(* CODESYS project IndraLogic.project

Project tree, tasks and I/O mapping:
  IndraMotionMlc1 : IndraControl XM2, Bosch Rexroth AG, order no. dependent on customer specific configuration, version 14.22.36.0
    application Application
      libraries: Linked List, 1.2.1.14 (Bosch Rexroth); MQTT Client, 2.3.8.14 (Bosch Rexroth)
      task PlcTask (cyclic, interval 10 ms, priority 5, watchdog 10 ms x 2) calls PlcProg
      task MotionTask (externalevent, external event EVENT_OP_MODE_MOTION_CYCLIC, priority 2, watchdog 4000 µs x 1) calls MotionProg
      function CheckBounds [ST]
      Symbols
      program PlcProg [ST]
      program MotionProg [ST]
      global variables MlcVarGlobal
      global variables IO
    S20_I_O : S20_I_O, Bosch Rexroth AG, version 14.22.10.1
    Sercos_III_Master : SercosIII Master, Rexroth, order no. 1, version 14.6.0.0
*)

// IndraMotionMlc1/Application/MlcVarGlobal
(* Automatically generated code by XLC/MLC. *)
(* Please don't edit, the code will be overwritten. For usercode use UserVarGlobal! *)
{attribute 'linkalways'}
{attribute 'analysis' := '-33'}
VAR_GLOBAL CONSTANT

(*Real axis "Axis1" with axis number 2*)
Axis1: AXIS_REF :=(CntrlNo:=LOCAL_CNTRL,AxisNo:=AXIS_2);


(*Probe 001*)
TouchProbe001: TOUCHPROBE_REF :=(CntrlNo:=LOCAL_CNTRL,TouchProbeNo:=TOUCHPROBE_1);

(*Probe 002*)
TouchProbe002: TOUCHPROBE_REF :=(CntrlNo:=LOCAL_CNTRL,TouchProbeNo:=TOUCHPROBE_2);

(*Probe 003*)
TouchProbe003: TOUCHPROBE_REF :=(CntrlNo:=LOCAL_CNTRL,TouchProbeNo:=TOUCHPROBE_3);

(*Probe 004*)
TouchProbe004: TOUCHPROBE_REF :=(CntrlNo:=LOCAL_CNTRL,TouchProbeNo:=TOUCHPROBE_4);

(*Probe 005*)
TouchProbe005: TOUCHPROBE_REF :=(CntrlNo:=LOCAL_CNTRL,TouchProbeNo:=TOUCHPROBE_5);

(*Probe 006*)
TouchProbe006: TOUCHPROBE_REF :=(CntrlNo:=LOCAL_CNTRL,TouchProbeNo:=TOUCHPROBE_6);

(*Probe 007*)
TouchProbe007: TOUCHPROBE_REF :=(CntrlNo:=LOCAL_CNTRL,TouchProbeNo:=TOUCHPROBE_7);

(*Probe 008*)
TouchProbe008: TOUCHPROBE_REF :=(CntrlNo:=LOCAL_CNTRL,TouchProbeNo:=TOUCHPROBE_8);

(*Probe 009*)
TouchProbe009: TOUCHPROBE_REF :=(CntrlNo:=LOCAL_CNTRL,TouchProbeNo:=TOUCHPROBE_9);

(*Probe 010*)
TouchProbe010: TOUCHPROBE_REF :=(CntrlNo:=LOCAL_CNTRL,TouchProbeNo:=TOUCHPROBE_10);

(*Probe 011*)
TouchProbe011: TOUCHPROBE_REF :=(CntrlNo:=LOCAL_CNTRL,TouchProbeNo:=TOUCHPROBE_11);

(*Probe 012*)
TouchProbe012: TOUCHPROBE_REF :=(CntrlNo:=LOCAL_CNTRL,TouchProbeNo:=TOUCHPROBE_12);

(*Probe 013*)
TouchProbe013: TOUCHPROBE_REF :=(CntrlNo:=LOCAL_CNTRL,TouchProbeNo:=TOUCHPROBE_13);

(*Probe 014*)
TouchProbe014: TOUCHPROBE_REF :=(CntrlNo:=LOCAL_CNTRL,TouchProbeNo:=TOUCHPROBE_14);

(*Probe 015*)
TouchProbe015: TOUCHPROBE_REF :=(CntrlNo:=LOCAL_CNTRL,TouchProbeNo:=TOUCHPROBE_15);

(*Probe 016*)
TouchProbe016: TOUCHPROBE_REF :=(CntrlNo:=LOCAL_CNTRL,TouchProbeNo:=TOUCHPROBE_16);

(*Probe 017*)
TouchProbe017: TOUCHPROBE_REF :=(CntrlNo:=LOCAL_CNTRL,TouchProbeNo:=TOUCHPROBE_17);

(*Probe 018*)
TouchProbe018: TOUCHPROBE_REF :=(CntrlNo:=LOCAL_CNTRL,TouchProbeNo:=TOUCHPROBE_18);

(*Probe 019*)
TouchProbe019: TOUCHPROBE_REF :=(CntrlNo:=LOCAL_CNTRL,TouchProbeNo:=TOUCHPROBE_19);

(*Probe 020*)
TouchProbe020: TOUCHPROBE_REF :=(CntrlNo:=LOCAL_CNTRL,TouchProbeNo:=TOUCHPROBE_20);

(*Probe 021*)
TouchProbe021: TOUCHPROBE_REF :=(CntrlNo:=LOCAL_CNTRL,TouchProbeNo:=TOUCHPROBE_21);

(*Probe 022*)
TouchProbe022: TOUCHPROBE_REF :=(CntrlNo:=LOCAL_CNTRL,TouchProbeNo:=TOUCHPROBE_22);

(*Probe 023*)
TouchProbe023: TOUCHPROBE_REF :=(CntrlNo:=LOCAL_CNTRL,TouchProbeNo:=TOUCHPROBE_23);

(*Probe 024*)
TouchProbe024: TOUCHPROBE_REF :=(CntrlNo:=LOCAL_CNTRL,TouchProbeNo:=TOUCHPROBE_24);

(*Probe 025*)
TouchProbe025: TOUCHPROBE_REF :=(CntrlNo:=LOCAL_CNTRL,TouchProbeNo:=TOUCHPROBE_25);

(*Probe 026*)
TouchProbe026: TOUCHPROBE_REF :=(CntrlNo:=LOCAL_CNTRL,TouchProbeNo:=TOUCHPROBE_26);

(*Probe 027*)
TouchProbe027: TOUCHPROBE_REF :=(CntrlNo:=LOCAL_CNTRL,TouchProbeNo:=TOUCHPROBE_27);

(*Probe 028*)
TouchProbe028: TOUCHPROBE_REF :=(CntrlNo:=LOCAL_CNTRL,TouchProbeNo:=TOUCHPROBE_28);

(*Probe 029*)
TouchProbe029: TOUCHPROBE_REF :=(CntrlNo:=LOCAL_CNTRL,TouchProbeNo:=TOUCHPROBE_29);

(*Probe 030*)
TouchProbe030: TOUCHPROBE_REF :=(CntrlNo:=LOCAL_CNTRL,TouchProbeNo:=TOUCHPROBE_30);

(*Probe 031*)
TouchProbe031: TOUCHPROBE_REF :=(CntrlNo:=LOCAL_CNTRL,TouchProbeNo:=TOUCHPROBE_31);

(*Probe 032*)
TouchProbe032: TOUCHPROBE_REF :=(CntrlNo:=LOCAL_CNTRL,TouchProbeNo:=TOUCHPROBE_32);

(*Probe 033*)
TouchProbe033: TOUCHPROBE_REF :=(CntrlNo:=LOCAL_CNTRL,TouchProbeNo:=TOUCHPROBE_33);

(*Probe 034*)
TouchProbe034: TOUCHPROBE_REF :=(CntrlNo:=LOCAL_CNTRL,TouchProbeNo:=TOUCHPROBE_34);

(*Probe 035*)
TouchProbe035: TOUCHPROBE_REF :=(CntrlNo:=LOCAL_CNTRL,TouchProbeNo:=TOUCHPROBE_35);

(*Probe 036*)
TouchProbe036: TOUCHPROBE_REF :=(CntrlNo:=LOCAL_CNTRL,TouchProbeNo:=TOUCHPROBE_36);

(*Probe 037*)
TouchProbe037: TOUCHPROBE_REF :=(CntrlNo:=LOCAL_CNTRL,TouchProbeNo:=TOUCHPROBE_37);

(*Probe 038*)
TouchProbe038: TOUCHPROBE_REF :=(CntrlNo:=LOCAL_CNTRL,TouchProbeNo:=TOUCHPROBE_38);

(*Probe 039*)
TouchProbe039: TOUCHPROBE_REF :=(CntrlNo:=LOCAL_CNTRL,TouchProbeNo:=TOUCHPROBE_39);

(*Probe 040*)
TouchProbe040: TOUCHPROBE_REF :=(CntrlNo:=LOCAL_CNTRL,TouchProbeNo:=TOUCHPROBE_40);

(*Probe 041*)
TouchProbe041: TOUCHPROBE_REF :=(CntrlNo:=LOCAL_CNTRL,TouchProbeNo:=TOUCHPROBE_41);

(*Probe 042*)
TouchProbe042: TOUCHPROBE_REF :=(CntrlNo:=LOCAL_CNTRL,TouchProbeNo:=TOUCHPROBE_42);

(*Probe 043*)
TouchProbe043: TOUCHPROBE_REF :=(CntrlNo:=LOCAL_CNTRL,TouchProbeNo:=TOUCHPROBE_43);

(*Probe 044*)
TouchProbe044: TOUCHPROBE_REF :=(CntrlNo:=LOCAL_CNTRL,TouchProbeNo:=TOUCHPROBE_44);

(*Probe 045*)
TouchProbe045: TOUCHPROBE_REF :=(CntrlNo:=LOCAL_CNTRL,TouchProbeNo:=TOUCHPROBE_45);

(*Probe 046*)
TouchProbe046: TOUCHPROBE_REF :=(CntrlNo:=LOCAL_CNTRL,TouchProbeNo:=TOUCHPROBE_46);

(*Probe 047*)
TouchProbe047: TOUCHPROBE_REF :=(CntrlNo:=LOCAL_CNTRL,TouchProbeNo:=TOUCHPROBE_47);

(*Probe 048*)
TouchProbe048: TOUCHPROBE_REF :=(CntrlNo:=LOCAL_CNTRL,TouchProbeNo:=TOUCHPROBE_48);

(*Probe 049*)
TouchProbe049: TOUCHPROBE_REF :=(CntrlNo:=LOCAL_CNTRL,TouchProbeNo:=TOUCHPROBE_49);

(*Probe 050*)
TouchProbe050: TOUCHPROBE_REF :=(CntrlNo:=LOCAL_CNTRL,TouchProbeNo:=TOUCHPROBE_50);

(*Probe 051*)
TouchProbe051: TOUCHPROBE_REF :=(CntrlNo:=LOCAL_CNTRL,TouchProbeNo:=TOUCHPROBE_51);

(*Probe 052*)
TouchProbe052: TOUCHPROBE_REF :=(CntrlNo:=LOCAL_CNTRL,TouchProbeNo:=TOUCHPROBE_52);

(*Probe 053*)
TouchProbe053: TOUCHPROBE_REF :=(CntrlNo:=LOCAL_CNTRL,TouchProbeNo:=TOUCHPROBE_53);

(*Probe 054*)
TouchProbe054: TOUCHPROBE_REF :=(CntrlNo:=LOCAL_CNTRL,TouchProbeNo:=TOUCHPROBE_54);

(*Probe 055*)
TouchProbe055: TOUCHPROBE_REF :=(CntrlNo:=LOCAL_CNTRL,TouchProbeNo:=TOUCHPROBE_55);

(*Probe 056*)
TouchProbe056: TOUCHPROBE_REF :=(CntrlNo:=LOCAL_CNTRL,TouchProbeNo:=TOUCHPROBE_56);

(*Probe 057*)
TouchProbe057: TOUCHPROBE_REF :=(CntrlNo:=LOCAL_CNTRL,TouchProbeNo:=TOUCHPROBE_57);

(*Probe 058*)
TouchProbe058: TOUCHPROBE_REF :=(CntrlNo:=LOCAL_CNTRL,TouchProbeNo:=TOUCHPROBE_58);

(*Probe 059*)
TouchProbe059: TOUCHPROBE_REF :=(CntrlNo:=LOCAL_CNTRL,TouchProbeNo:=TOUCHPROBE_59);

(*Probe 060*)
TouchProbe060: TOUCHPROBE_REF :=(CntrlNo:=LOCAL_CNTRL,TouchProbeNo:=TOUCHPROBE_60);

(*Probe 061*)
TouchProbe061: TOUCHPROBE_REF :=(CntrlNo:=LOCAL_CNTRL,TouchProbeNo:=TOUCHPROBE_61);

(*Probe 062*)
TouchProbe062: TOUCHPROBE_REF :=(CntrlNo:=LOCAL_CNTRL,TouchProbeNo:=TOUCHPROBE_62);

(*Probe 063*)
TouchProbe063: TOUCHPROBE_REF :=(CntrlNo:=LOCAL_CNTRL,TouchProbeNo:=TOUCHPROBE_63);

(*Probe 064*)
TouchProbe064: TOUCHPROBE_REF :=(CntrlNo:=LOCAL_CNTRL,TouchProbeNo:=TOUCHPROBE_64);

(*Probe 065*)
TouchProbe065: TOUCHPROBE_REF :=(CntrlNo:=LOCAL_CNTRL,TouchProbeNo:=TOUCHPROBE_65);

(*Probe 066*)
TouchProbe066: TOUCHPROBE_REF :=(CntrlNo:=LOCAL_CNTRL,TouchProbeNo:=TOUCHPROBE_66);

(*Probe 067*)
TouchProbe067: TOUCHPROBE_REF :=(CntrlNo:=LOCAL_CNTRL,TouchProbeNo:=TOUCHPROBE_67);

(*Probe 068*)
TouchProbe068: TOUCHPROBE_REF :=(CntrlNo:=LOCAL_CNTRL,TouchProbeNo:=TOUCHPROBE_68);

(*Probe 069*)
TouchProbe069: TOUCHPROBE_REF :=(CntrlNo:=LOCAL_CNTRL,TouchProbeNo:=TOUCHPROBE_69);

(*Probe 070*)
TouchProbe070: TOUCHPROBE_REF :=(CntrlNo:=LOCAL_CNTRL,TouchProbeNo:=TOUCHPROBE_70);

(*Probe 071*)
TouchProbe071: TOUCHPROBE_REF :=(CntrlNo:=LOCAL_CNTRL,TouchProbeNo:=TOUCHPROBE_71);

(*Probe 072*)
TouchProbe072: TOUCHPROBE_REF :=(CntrlNo:=LOCAL_CNTRL,TouchProbeNo:=TOUCHPROBE_72);

(*Probe 073*)
TouchProbe073: TOUCHPROBE_REF :=(CntrlNo:=LOCAL_CNTRL,TouchProbeNo:=TOUCHPROBE_73);

(*Probe 074*)
TouchProbe074: TOUCHPROBE_REF :=(CntrlNo:=LOCAL_CNTRL,TouchProbeNo:=TOUCHPROBE_74);

(*Probe 075*)
TouchProbe075: TOUCHPROBE_REF :=(CntrlNo:=LOCAL_CNTRL,TouchProbeNo:=TOUCHPROBE_75);

(*Probe 076*)
TouchProbe076: TOUCHPROBE_REF :=(CntrlNo:=LOCAL_CNTRL,TouchProbeNo:=TOUCHPROBE_76);

(*Probe 077*)
TouchProbe077: TOUCHPROBE_REF :=(CntrlNo:=LOCAL_CNTRL,TouchProbeNo:=TOUCHPROBE_77);

(*Probe 078*)
TouchProbe078: TOUCHPROBE_REF :=(CntrlNo:=LOCAL_CNTRL,TouchProbeNo:=TOUCHPROBE_78);

(*Probe 079*)
TouchProbe079: TOUCHPROBE_REF :=(CntrlNo:=LOCAL_CNTRL,TouchProbeNo:=TOUCHPROBE_79);

(*Probe 080*)
TouchProbe080: TOUCHPROBE_REF :=(CntrlNo:=LOCAL_CNTRL,TouchProbeNo:=TOUCHPROBE_80);

(*Probe 081*)
TouchProbe081: TOUCHPROBE_REF :=(CntrlNo:=LOCAL_CNTRL,TouchProbeNo:=TOUCHPROBE_81);

(*Probe 082*)
TouchProbe082: TOUCHPROBE_REF :=(CntrlNo:=LOCAL_CNTRL,TouchProbeNo:=TOUCHPROBE_82);

(*Probe 083*)
TouchProbe083: TOUCHPROBE_REF :=(CntrlNo:=LOCAL_CNTRL,TouchProbeNo:=TOUCHPROBE_83);

(*Probe 084*)
TouchProbe084: TOUCHPROBE_REF :=(CntrlNo:=LOCAL_CNTRL,TouchProbeNo:=TOUCHPROBE_84);

(*Probe 085*)
TouchProbe085: TOUCHPROBE_REF :=(CntrlNo:=LOCAL_CNTRL,TouchProbeNo:=TOUCHPROBE_85);

(*Probe 086*)
TouchProbe086: TOUCHPROBE_REF :=(CntrlNo:=LOCAL_CNTRL,TouchProbeNo:=TOUCHPROBE_86);

(*Probe 087*)
TouchProbe087: TOUCHPROBE_REF :=(CntrlNo:=LOCAL_CNTRL,TouchProbeNo:=TOUCHPROBE_87);

(*Probe 088*)
TouchProbe088: TOUCHPROBE_REF :=(CntrlNo:=LOCAL_CNTRL,TouchProbeNo:=TOUCHPROBE_88);

(*Probe 089*)
TouchProbe089: TOUCHPROBE_REF :=(CntrlNo:=LOCAL_CNTRL,TouchProbeNo:=TOUCHPROBE_89);

(*Probe 090*)
TouchProbe090: TOUCHPROBE_REF :=(CntrlNo:=LOCAL_CNTRL,TouchProbeNo:=TOUCHPROBE_90);

(*Probe 091*)
TouchProbe091: TOUCHPROBE_REF :=(CntrlNo:=LOCAL_CNTRL,TouchProbeNo:=TOUCHPROBE_91);

(*Probe 092*)
TouchProbe092: TOUCHPROBE_REF :=(CntrlNo:=LOCAL_CNTRL,TouchProbeNo:=TOUCHPROBE_92);

(*Probe 093*)
TouchProbe093: TOUCHPROBE_REF :=(CntrlNo:=LOCAL_CNTRL,TouchProbeNo:=TOUCHPROBE_93);

(*Probe 094*)
TouchProbe094: TOUCHPROBE_REF :=(CntrlNo:=LOCAL_CNTRL,TouchProbeNo:=TOUCHPROBE_94);

(*Probe 095*)
TouchProbe095: TOUCHPROBE_REF :=(CntrlNo:=LOCAL_CNTRL,TouchProbeNo:=TOUCHPROBE_95);

(*Probe 096*)
TouchProbe096: TOUCHPROBE_REF :=(CntrlNo:=LOCAL_CNTRL,TouchProbeNo:=TOUCHPROBE_96);

(*Probe 097*)
TouchProbe097: TOUCHPROBE_REF :=(CntrlNo:=LOCAL_CNTRL,TouchProbeNo:=TOUCHPROBE_97);

(*Probe 098*)
TouchProbe098: TOUCHPROBE_REF :=(CntrlNo:=LOCAL_CNTRL,TouchProbeNo:=TOUCHPROBE_98);

(*Probe 099*)
TouchProbe099: TOUCHPROBE_REF :=(CntrlNo:=LOCAL_CNTRL,TouchProbeNo:=TOUCHPROBE_99);

(*Probe 100*)
TouchProbe100: TOUCHPROBE_REF :=(CntrlNo:=LOCAL_CNTRL,TouchProbeNo:=TOUCHPROBE_100);

END_VAR

// IndraMotionMlc1/Application/IO
{attribute 'qualified_only'}
VAR_GLOBAL
	
END_VAR

// IndraMotionMlc1/Application/PlcProg
PROGRAM PlcProg
VAR
	rVelocity		:	REAL;
	bIsAxisEnabled 	: 	BOOL;
	pwrOn			: 	MC_Power;
	moveVel			:	MC_MoveVelocity;
	stopAxis		:	MC_Stop;
END_VAR

VAR
	mqttClient 			: MQTTClientFB;
	mqttStatusPublish 	: MQTTPublishFB;
	mqttSubscribe 		: MQTTSubscribeFB;
	mqttString 			: MQTTGetStringFB;
	
	sMQTT_TOPIC_SERVO_CMD 	: STRING :='SERVO/CMD';
	sMQTT_TOPIC_CONNECTION 	: STRING :='SERVO/CONNECTION';
	
	sPayloads				: STRING:='ONLINE';
	
	sMES 			: STRING;
	sCMD 			: STRING;
	rVel			: REAL;
	
	tonTimer		: TON;
	tonTimerStop	: TON;
	tonTimerOFF		: TON;
	tonTimerBOFF	: TON;
//	Off				: BOOL;
END_VAR

mqttClient(
	Enable:= TRUE , 
	IPAddress:='192.168.99.100', 
	Port:= 1883 , 
	ConnectionTimeout:= , 
	KeepAlive:= 10, 
	ClientID:= 'plcClient', 
	Username:= , 
	Password:= , 
	LastWillRetain:= , 
	LastWillTopic:= sMQTT_TOPIC_CONNECTION , 
	LastWillMessage:= 'OFFLINE', 
	LastWillQos:= , 
	TCPConnected=> , 
	Connected=> , 
	Socket=> , 
	PubAckID=> , 
	ErrorCode=> , 
	ErrorInfo=> , 
	ConnectionState=> , 
	SubscribedDataRecvd=> );

mqttSubscribe(
	Enable:= mqttClient.Connected, 
	Post:= tonTimer.Q , 
	Topic:= sMQTT_TOPIC_SERVO_CMD, 
	QoS:= ,  
	ConnectionHandle:= ADR(mqttClient), 
	ErrorCode=> , 
	RunningState=> , 
	Complete=> , 
	Retries=> );

mqttString(
	Enable:= mqttSubscribe.Complete, 
	Topic:= sMQTT_TOPIC_SERVO_CMD, 
	Prefix:= , 
	Enabled=> , 
	Output=> sMES, 
	Done=> );	
	
mqttStatusPublish(
	Enable:= mqttClient.Connected, 
	Post:= tonTimer.Q , 
	Retained:= , 
	QoS:= , 
	Topic:= sMQTT_TOPIC_CONNECTION , 
	Payload:= ADR(sPayloads), 
	DataLength:= INT_TO_UINT(len(sPayloads)) , 
	ConnectionHandle:= ADR(mqttClient) , 
	ErrorCode=> , 
	RunningState=> );
	
tonTimer(IN:= mqttClient.Connected , PT:= T#1S , Q=> , ET=> );
tonTimerStop(IN:= NOT mqttClient.Connected , PT:= T#3S , Q=> , ET=> );
tonTimerOFF(IN:= , PT:= T#0.1S , Q=> , ET=> );
tonTimerBOFF(IN:= , PT:= T#0.1S , Q=> , ET=> );

IF mqttString.Done THEN
	sCMD := LEFT(sMES,2);
	rVel := STRING_TO_REAL(DELETE(sMes,2,1));
	IF sMES = 'RUN' OR sMES = 'run' THEN
		pwrOn.Enable := TRUE;
		stopAxis.Execute := FALSE;
	ELSIF sCMD = 'X' THEN
		moveVel.Execute := FALSE ;
	ELSIF sCMD = 'RV' AND rVel > 0 AND rVel < 500 THEN
		rVelocity := rVel;
		moveVel.Execute := TRUE ;
	ELSIF sCMD = 'LV' AND rVel > 0 AND rVel < 500 THEN
		rVelocity := -1 * rVel;
		moveVel.Execute := TRUE ;
	ELSIF sMES = 'STOP' OR sMES = 'stop' THEN
		stopAxis.Execute := TRUE;
		moveVel.Execute := FALSE;
		rVelocity := 0;
	ELSIF sMES = 'START' OR sMES = 'start' THEN
		stopAxis.Execute := FALSE;
	ELSIF sMES = 'OFF' OR sMES = 'off' THEN
		stopAxis.Execute := TRUE;
		tonTimerOFF.IN := TRUE ;
	END_IF
END_IF
IF tonTimerOFF.Q = TRUE THEN
	stopAxis.Execute := FALSE;
	tonTimerBOFF.IN := TRUE ;
END_IF
 
IF tonTimerBOFF.Q = TRUE THEN
	pwrOn.Enable := FALSE;
	tonTimerBOFF.IN := FALSE;
	tonTimerOFF.IN := FALSE;
END_IF

pwrOn(
	Enable:= ,
	Status=> bIsAxisEnabled, 
	Error=> , 
	ErrorID=> , 
	ErrorIdent=> , 
	Axis:= Axis1);

moveVel(
	Execute:= , 
	Velocity:= rVelocity, 
	Acceleration:= 1000, 
	Deceleration:= 1000, 
	InVelocity=> , 
	Active=> , 
	CommandAborted=> , 
	Error=> , 
	ErrorID=> , 
	ErrorIdent=> , 
	Axis:= Axis1 );

stopAxis(
	Execute:= , 
	Deceleration:= 1000, 
	Done=> , 
	Active=> , 
	CommandAborted=> , 
	Error=> , 
	ErrorID=> , 
	ErrorIdent=> , 
	Axis:= Axis1);

END_PROGRAM

// IndraMotionMlc1/Application/MotionProg
PROGRAM MotionProg
VAR
END_VAR

END_PROGRAM

// IndraMotionMlc1/Application/CheckBounds
(*
General Header
----------------------------------------------------------------------------------------------
Short description      : Function to check access to array within valid bounds.
                         After inserting/removing this function, no online-change will be possible! A complete download will be necessary!
Version                : 14.1.0.0
Author                 : DC-IA/EAM3 (MD)
Date                   : 2015-01-12
Company                : Bosch Rexroth AG
Target                 : IndraLogic XLC/MLC
Functional description : This function will be called implicitly before the read/write access
                         to arrays takes places.
                         The index of the subsequent array accesses is checked for valid
                         limits.
                         In case of invalid access, an error is entered in the diagnostic
                         logbook and the application is stopped due to an access violation to
                         avoid machine damage.
                         In this case, check the callstack (menu Debug/Callstack) and modify
                         the faulty logic. 
Handling specials      : This function increases the cycle time of all IEC-tasks using array
                         accesses. 
                         The increase depends on the number of the read/write accesses to
                         arrays.
                         After inserting/removing this function, no online-change will be possible! 
                         A complete download will be necessary!
						 This is an exemplary implementation of the function. 
                         The implementation has to be adjusted to your application/machine.
						 Per default, the PLC-Task will generate an access violation which leads to
                         an application stop and a F5-error with error reaction respectively.
                         Please verify whether this default behaviour can damage your machine 
                         or lead to a complex recommissioning. 
                         In this case, adapt the error reaction to your application.
						 
                         If your application isn't too time-critical, you should leave this function 
						 while commissioning the machine and production in your application.  
                         If you remove this funciton, ensure that your code is faultless.
                         
                         Do not modify the declaration of this function! 
                         Do not change the attributes above the function header!
----------------------------------------------------------------------------------------------
*)
{attribute 'check_bounds'}
{attribute 'no_check'}
{attribute 'signature_flag' := '1073741824'}
FUNCTION CheckBounds : DINT
VAR_INPUT
	index, lower, upper: DINT;
END_VAR
VAR
	{attribute 'hide'}
	bByte: BYTE;
	ptNull: POINTER TO BYTE :=0;
	errstr: STRING;
	
END_VAR

(*************************************************************
This function was generated by the 'check array access'
option of the controllers 'properties' dialog box.
If you delete this comment, the 'check array access' option
of the controllers 'properties' dialog box will be removed.
**************************************************************)
    (**************************************************************************************************)
    (* The implementation has to be adjusted to your application/machine.                             *)
    (* This is an exemplary implementation of the function.                                           *)
    (* Per default, an access violation is generated to avoid machine damage                          *)
    (* Check the Call Stack (menu Debug/Callstack) and modify the faulty logic!                       *)
    (**************************************************************************************************)

IF  index < lower THEN 
	errstr:= 'CheckBounds: Lower arrayindex ';
	errstr:=CONCAT(STR1:=errstr  , STR2:= DINT_TO_STRING(lower));
	errstr:=CONCAT(STR1:=errstr  , STR2:= ' underrunned by ');
	errstr:=CONCAT(STR1:=errstr  , STR2:= DINT_TO_STRING(index));
//  This pragma may be removed: 
	{info 'CheckBounds: Please implement your own error reaction below'}
//  EXAMPLE 1 (default): 
//  Set a F0-Error into the diagnostic- and error memory
//  Triggering an access violation --> Application will be stopped and leads to a F5-Error

  ML_SetDiagEntry(
	Severity:= E_LOG_SEVERITY.ERROR, 
	Class:= E_LOG_CLASS.CLASS_0, 
	Facility:= E_LOG_FACILITY.USER, 
	Code:= 0, 
	Text:= ADR(errstr));

	bByte:=ptNull^;(*triggering an access violation *)

// EXAMPLE 2:
// Limit the faulty index to the lower index 
//     -> no memory will be overwritten
//     -> Keep PLC-task and motion running
// Set a E0-Warning into the diagnostic- and error memory
// NOTE: There is still an implementation error in your application code!

//  ML_SetDiagEntry(
//	Severity:= E_LOG_SEVERITY.WARNING, 
//	Class:= E_LOG_CLASS.CLASS_0, 
//	Facility:= E_LOG_FACILITY.USER, 
//	Code:= 0, 
//	Text:= ADR(errstr));
// 
//	CheckBounds := lower; //access to the lower index only 
//  return;
	
ELSIF  index > upper THEN
	errstr:= 'CheckBounds: Higher arrayindex ';
	errstr:=CONCAT(STR1:=errstr  , STR2:= DINT_TO_STRING(upper));
	errstr:=CONCAT(STR1:=errstr  , STR2:= ' overrunned by ');
	errstr:=CONCAT(STR1:=errstr  , STR2:= DINT_TO_STRING(index));

//  this pragma may be removed: 
	{info 'CheckBounds: Please implement your own error reaction below'}
//  example 1 (default): 
//  set a F0-Error into the diagnostic- and error memory
//  triggering an access violation --> Application will be stopped and leads to a F5-Error

  ML_SetDiagEntry(
	Severity:= E_LOG_SEVERITY.ERROR, 
	Class:= E_LOG_CLASS.CLASS_0, 
	Facility:= E_LOG_FACILITY.USER, 
	Code:= 0, 
	Text:= ADR(errstr));

	bByte:=ptNull^;(*triggering an access violation *)

//example 2:
// Limit the faulty index to the upper index 
//     -> no memory will be overwritten
//     -> Keep PLC-task and motion running
// Set a E0-Warning into the diagnostic- and error memory
// NOTE: There is still an implementation error in your application code!

//  ML_SetDiagEntry(
//	Severity:= E_LOG_SEVERITY.WARNING, 
//	Class:= E_LOG_CLASS.CLASS_0, 
//	Facility:= E_LOG_FACILITY.USER, 
//	Code:= 0, 
//	Text:= ADR(errstr));
// 
//	CheckBounds := upper; //access to the upper index only 
//  return;

ELSE // access to array is ok  
	CheckBounds := index;
END_IF

END_FUNCTION
